// Fluent builder interface for composing log entries.
// Obtain an instance via F_Log() or FB_Log.Log(), chain methods, and call CreateLog() to emit.
INTERFACE I_WithContext EXTENDS I_Logger

// Attaches context properties to this log entry.
// Use F_Context() to create a temporary context, or pass an FB_ContextBuilder instance.
METHOD WithContext : I_Logger
VAR_INPUT
	iContextBuilder	: I_ContextBuilder;
END_VAR
END_METHOD

END_INTERFACE

(* stored: Version 1.1.0.1, ProductVersion 3.1.4026.17
   Itf I_WithContext: Id {449596c7-422a-0b36-3e3d-0d838674fb28}
   Method WithContext: Id {8f3ae027-986c-0245-1eea-dea78c28d234} *)
